Fanuc KAREL source: kb00064.KL

PROGRAM KB00064
%NOLOCKGROUP
VAR
P1 : STRING[80];P2 : STRING[80];P3:INTEGER
BEGIN
--
--
P1='A'
P2='A'
P3=1
DET_WINDOW(P1,P2,P3)
END KB00064
